(* IEC 61131-3 sources: STruCpp/examples, 6 files *)

(* ---- counter.st ---- *)
(*
 * Counter Example
 *
 * A simple up/down counter with reset functionality.
 * Demonstrates basic arithmetic and conditional logic.
 *)

FUNCTION_BLOCK Counter
  VAR_INPUT
    countUp : BOOL;    (* Count up on rising edge *)
    countDown : BOOL;  (* Count down on rising edge *)
    reset : BOOL;      (* Reset counter to zero *)
    maxValue : INT := 100;  (* Maximum count value *)
    minValue : INT := 0;    (* Minimum count value *)
  END_VAR

  VAR_OUTPUT
    count : INT;       (* Current count value *)
    atMax : BOOL;      (* TRUE when at maximum *)
    atMin : BOOL;      (* TRUE when at minimum *)
  END_VAR

  VAR
    prevUp : BOOL;     (* Previous state of countUp *)
    prevDown : BOOL;   (* Previous state of countDown *)
  END_VAR

  (* Reset handling *)
  IF reset THEN
    count := 0;
  ELSE
    (* Count up on rising edge *)
    IF countUp AND NOT prevUp THEN
      IF count < maxValue THEN
        count := count + 1;
      END_IF;
    END_IF;

    (* Count down on rising edge *)
    IF countDown AND NOT prevDown THEN
      IF count > minValue THEN
        count := count - 1;
      END_IF;
    END_IF;
  END_IF;

  (* Update edge detection *)
  prevUp := countUp;
  prevDown := countDown;

  (* Update status outputs *)
  atMax := count >= maxValue;
  atMin := count <= minValue;

END_FUNCTION_BLOCK

(* ---- pid_controller.st ---- *)
(*
 * PID Controller Example
 *
 * A basic PID (Proportional-Integral-Derivative) controller
 * function block for process control applications.
 *)

FUNCTION_BLOCK PID_Controller
  VAR_INPUT
    setpoint : REAL;      (* Desired value *)
    processValue : REAL;  (* Measured value *)
    kp : REAL := 1.0;     (* Proportional gain *)
    ki : REAL := 0.1;     (* Integral gain *)
    kd : REAL := 0.01;    (* Derivative gain *)
    dt : REAL := 0.1;     (* Sample time in seconds *)
    outMin : REAL := 0.0; (* Minimum output *)
    outMax : REAL := 100.0; (* Maximum output *)
    enable : BOOL := TRUE; (* Enable controller *)
    reset : BOOL;         (* Reset integrator *)
  END_VAR

  VAR_OUTPUT
    output : REAL;        (* Controller output *)
    error : REAL;         (* Current error *)
  END_VAR

  VAR
    integral : REAL;      (* Integral accumulator *)
    prevError : REAL;     (* Previous error for derivative *)
    derivative : REAL;    (* Derivative term *)
    pTerm : REAL;         (* Proportional term *)
    iTerm : REAL;         (* Integral term *)
    dTerm : REAL;         (* Derivative term *)
  END_VAR

  (* Reset integrator if requested *)
  IF reset THEN
    integral := 0.0;
    prevError := 0.0;
    output := 0.0;
  ELSIF enable THEN
    (* Calculate error *)
    error := setpoint - processValue;

    (* Proportional term *)
    pTerm := kp * error;

    (* Integral term with anti-windup *)
    integral := integral + (error * dt);
    iTerm := ki * integral;

    (* Derivative term *)
    derivative := (error - prevError) / dt;
    dTerm := kd * derivative;

    (* Calculate output *)
    output := pTerm + iTerm + dTerm;

    (* Clamp output to limits *)
    IF output > outMax THEN
      output := outMax;
      (* Anti-windup: prevent integral from growing *)
      IF error > 0.0 THEN
        integral := integral - (error * dt);
      END_IF;
    ELSIF output < outMin THEN
      output := outMin;
      (* Anti-windup: prevent integral from shrinking *)
      IF error < 0.0 THEN
        integral := integral - (error * dt);
      END_IF;
    END_IF;

    (* Save error for next iteration *)
    prevError := error;
  END_IF;

END_FUNCTION_BLOCK

(* ---- unity_conveyor_controller.st ---- *)
(*
 * Unity Conveyor Controller Example
 *
 * Purpose:
 * - Run as a virtual PLC controller for a Unity digital twin.
 * - Inputs/outputs are plain BOOL tags that map cleanly to Unity C#.
 *
 * Scan assumptions:
 * - Controller cycle is 10 ms.
 * - Jam timeout is 2.0 s => 200 cycles.
 *)

FUNCTION_BLOCK UnityConveyorController
  VAR_INPUT
    StartPB : BOOL;      (* Start pushbutton *)
    StopPB : BOOL;       (* Stop pushbutton *)
    JamSensor : BOOL;    (* True while conveyor is jammed *)
    ResetPB : BOOL;      (* Reset alarm pushbutton *)
    EStopOK : BOOL;      (* Emergency chain healthy *)
    GuardDoorClosed : BOOL; (* Safety guard status *)
  END_VAR

  VAR_OUTPUT
    MotorOn : BOOL;      (* Conveyor motor command *)
    Alarm : BOOL;        (* General alarm status *)
    JamActive : BOOL;    (* Jam timeout reached *)
    Ready : BOOL;        (* Machine can start/run *)
  END_VAR

  VAR
    runRequest : BOOL;
    jamCounter : UINT;
    safetyOK : BOOL;
  END_VAR

  safetyOK := EStopOK AND GuardDoorClosed;
  Ready := safetyOK AND NOT Alarm;

  (* Latch run command *)
  IF StartPB AND Ready THEN
    runRequest := TRUE;
  END_IF;

  (* Stop conditions clear run request *)
  IF StopPB OR NOT safetyOK OR JamActive THEN
    runRequest := FALSE;
  END_IF;

  (* Jam monitoring while conveyor is requested to run *)
  IF runRequest AND JamSensor THEN
    IF jamCounter < 200 THEN
      jamCounter := jamCounter + 1;
    END_IF;
  ELSE
    jamCounter := 0;
  END_IF;

  IF jamCounter >= 200 THEN
    JamActive := TRUE;
  END_IF;

  (* Alarm handling *)
  IF JamActive OR NOT safetyOK THEN
    Alarm := TRUE;
  END_IF;

  IF ResetPB AND safetyOK AND NOT JamSensor THEN
    JamActive := FALSE;
    Alarm := FALSE;
    jamCounter := 0;
  END_IF;

  MotorOn := runRequest AND safetyOK AND NOT Alarm;
END_FUNCTION_BLOCK

(* ---- blink.st ---- *)
(*
 * Blink Example
 *
 * A simple program that toggles an output at a fixed interval.
 * This is the "Hello World" of PLC programming.
 *)

PROGRAM Blink
  VAR
    output AT %QX0.0 : BOOL;  (* Output to toggle *)
    timer : TON;               (* On-delay timer *)
    interval : TIME := T#500ms; (* Blink interval *)
  END_VAR

  (* Toggle output when timer expires *)
  timer(IN := NOT timer.Q, PT := interval);

  IF timer.Q THEN
    output := NOT output;
  END_IF;

END_PROGRAM

(* ---- motor_control.st ---- *)
(*
 * Motor Control Example
 *
 * A simple motor control program with start/stop buttons,
 * emergency stop, and overload protection.
 *)

PROGRAM MotorControl
  VAR
    (* Inputs *)
    startButton AT %IX0.0 : BOOL;   (* Start pushbutton *)
    stopButton AT %IX0.1 : BOOL;    (* Stop pushbutton *)
    emergencyStop AT %IX0.2 : BOOL; (* Emergency stop (NC) *)
    overloadTrip AT %IX0.3 : BOOL;  (* Thermal overload relay *)

    (* Outputs *)
    motorContactor AT %QX0.0 : BOOL; (* Motor contactor output *)
    runningLamp AT %QX0.1 : BOOL;    (* Running indicator lamp *)
    faultLamp AT %QX0.2 : BOOL;      (* Fault indicator lamp *)

    (* Internal variables *)
    motorRunning : BOOL;  (* Motor running state *)
    faultActive : BOOL;   (* Fault condition active *)
  END_VAR

  (* Check for fault conditions *)
  faultActive := NOT emergencyStop OR overloadTrip;

  (* Motor control logic *)
  IF faultActive THEN
    (* Stop motor on any fault *)
    motorRunning := FALSE;
  ELSIF stopButton THEN
    (* Stop button pressed *)
    motorRunning := FALSE;
  ELSIF startButton AND NOT motorRunning THEN
    (* Start button pressed and motor not running *)
    motorRunning := TRUE;
  END_IF;

  (* Update outputs *)
  motorContactor := motorRunning;
  runningLamp := motorRunning;
  faultLamp := faultActive;

END_PROGRAM

(* ---- unity_conveyor_controller_tests.st ---- *)
TEST 'Conveyor starts when safety is healthy'
  VAR ctrl : UnityConveyorController; END_VAR
  ctrl.EStopOK := TRUE;
  ctrl.GuardDoorClosed := TRUE;
  ctrl.StartPB := TRUE;
  ctrl();
  ASSERT_TRUE(ctrl.MotorOn);
  ASSERT_FALSE(ctrl.Alarm);
END_TEST

TEST 'Stop button stops conveyor'
  VAR ctrl : UnityConveyorController; END_VAR
  ctrl.EStopOK := TRUE;
  ctrl.GuardDoorClosed := TRUE;
  ctrl.StartPB := TRUE;
  ctrl();
  ASSERT_TRUE(ctrl.MotorOn);

  ctrl.StartPB := FALSE;
  ctrl.StopPB := TRUE;
  ctrl();
  ASSERT_FALSE(ctrl.MotorOn);
END_TEST

TEST 'Jam alarm trips after 2 seconds at 10 ms scan'
  VAR
    ctrl : UnityConveyorController;
    i : UINT;
  END_VAR

  ctrl.EStopOK := TRUE;
  ctrl.GuardDoorClosed := TRUE;
  ctrl.StartPB := TRUE;
  ctrl();
  ctrl.StartPB := FALSE;
  ASSERT_TRUE(ctrl.MotorOn);

  ctrl.JamSensor := TRUE;
  FOR i := 1 TO 200 DO
    ctrl();
  END_FOR;

  ASSERT_TRUE(ctrl.JamActive);
  ASSERT_TRUE(ctrl.Alarm);
  ASSERT_FALSE(ctrl.MotorOn);
END_TEST

TEST 'Reset clears jam alarm when jam is removed'
  VAR
    ctrl : UnityConveyorController;
    i : UINT;
  END_VAR

  ctrl.EStopOK := TRUE;
  ctrl.GuardDoorClosed := TRUE;
  ctrl.StartPB := TRUE;
  ctrl();
  ctrl.StartPB := FALSE;
  ctrl.JamSensor := TRUE;

  FOR i := 1 TO 200 DO
    ctrl();
  END_FOR;

  ASSERT_TRUE(ctrl.Alarm);

  ctrl.JamSensor := FALSE;
  ctrl.ResetPB := TRUE;
  ctrl();
  ASSERT_FALSE(ctrl.Alarm);
  ASSERT_FALSE(ctrl.JamActive);
  ASSERT_FALSE(ctrl.MotorOn);

  ctrl.ResetPB := FALSE;
  ctrl.StartPB := TRUE;
  ctrl();
  ASSERT_TRUE(ctrl.MotorOn);
END_TEST
